# EPICS substitutions: EUROTHRM/EUROTHRM-IOC-01App/Db/devEurothrmA02.substitutions
# Note: this file is generated by generate_substitutions.py
file devEurothrm.template {
pattern { P, GAD, LAD, MODBUS_PV, MODBUS_SP, MODBUS_P, MODBUS_I, MODBUS_D, MODBUS_HS, MODBUS_LS, MODBUS_AT, MODBUS_HO, MODBUS_OP }
{ "\$(P)", "0", "2", "1025", "1026", "1030", "1032", "1033", "1135", "1136", "1294", "1054", "1027" }
}
